FUNCTION_BLOCK RunLifterCelluar EXTENDS RunUnitGeneric
VAR_INPUT
END_VAR
VAR_OUTPUT
END_VAR
VAR	
	//actuator
	//axis
	Axis : POINTER TO RunAxis;
	//cylinder
	Cylinder : POINTER TO RunCylinder;
	
	//lifter
	ptCommandLifterHit : POINTER TO ParameterSet; // raise to hit
	ptCommandLifterRelease : POINTER TO ParameterSet; //release
	ptCommandLifterWorking : POINTER TO ParameterSet; //lift carrier to working position
	//sensor
	ptObstacleSensorStatus : POINTER TO BOOL; //fibers
	ptReachSensorStatus : POINTER TO BOOL; //approximities
	//slot status
	ptPreivousSlotValid : POINTER TO BOOL;
	
END_VAR


CASE State OF
	0:
	//if execute flag on
	bSerialTransition := Axis^.ExecuteParameter(ptBlock:=ptCommandLifterHit);
	1:
	//once reach sensor detected , n
	bSerialTransition := ptReachSensorStatus^;
	2:
	//hold
	bSerialTransition := Cylinder^.Execute(eCylinderCommands.COMMAND_B);
	3:
	//to working position
	bSerialTransition := Axis^.ExecuteParameter(ptCommandLifterWorking);
	4:
	//if release flag on
	bSerialTransition := Axis^.ExecuteParameter(ptCommandLifterHit);
	5:
	//release holder
	bSerialTransition := Cylinder^.Execute(eCylinderCommands.COMMAND_A);
	6:
	IF Axis^.ExecuteParameter(ptCommandLifterRelease) THEN
		NextState := 0;
	END_IF
END_CASE

METHOD CheckReach : BOOL
VAR_INPUT
END_VAR
VAR_OUTPUT
	//neither Done nor Error : Transition
	Done:BOOL;	//successfully
END_VAR
//TODO , slot valid and reach sensor status or not slot valid
Done := ptReachSensorStatus^;
END_METHOD

METHOD FB_init : BOOL
VAR_INPUT
	bInitRetains : BOOL; // if TRUE, the retain variables are initialized (warm start / cold start)
	bInCopyCode : BOOL;  // if TRUE, the instance afterwards gets moved into the copy code (online change)
END_VAR
//initializing , link related commandblock/sensor/cylinder
END_METHOD

METHOD Initialize : BOOL
VAR_INPUT
END_VAR

CASE State OF
	0:
	bSerialTransition:=Cylinder^.Execute(eCylinderCommands.COMMAND_A);
	1:
	IF Axis^.ExecuteParameter(ptCommandLifterRelease) THEN
		NextState := 16#FF;	
	END_IF
END_CASE

Initialize := SUPER^.Initialize(); //call base method
END_METHOD

METHOD RaiseStopper : BOOL
VAR_INPUT
END_VAR
VAR_OUTPUT
	//neither Done nor Error : Transition
	Done:BOOL;	//successfully
END_VAR
VAR
END_VAR
//condition to execute :
//previous slot is valid and
//execute and
//obstacle not existed

//plus my slot is empty
Axis^.ExecuteCommandBlock(
ptBlock:= ptCommandLifterHit, 
execute:= TRUE,//ptPreivousSlotValid^ AND NOT ptObstacleSensorStatus^, 
bufferIndex:=1,
done=> );	

//Done:
//no need to raise
//or need to raise and successfully done	
//Done :=  (ptPreivousSlotValid^ AND ptAxis^.ExecuteCommandBlock.done) OR (NOT ptPreivousSlotValid^);
Done :=done;
END_METHOD

METHOD ReleaseStopper : BOOL
VAR_INPUT
END_VAR
VAR_OUTPUT
	Done:BOOL;	//successfully
END_VAR
Axis^.ExecuteCommandBlock(
ptBlock:= ptCommandLifterRelease, 
execute:= TRUE,//ptPreivousSlotValid^ AND NOT ptObstacleSensorStatus^, 
bufferIndex:=1,
done=> Done);
END_METHOD

END_FUNCTION_BLOCK

(* stored: Version 1.1.0.1, ProductVersion 3.1.4022.10
   POU RunLifterCelluar: Id {8e8fc5f3-47f1-4079-a3ab-596940aadfbf}, SpecialFunc None
   Method CheckReach: Id {67fa871c-5756-49a6-b887-c646b2442d16}
   Method FB_init: Id {a4e43bb3-b045-4468-b1e1-3d38f2c0d86a}
   Method Initialize: Id {21db5a00-f7a1-4530-94de-d799f1b897b9}
   Method RaiseStopper: Id {54b07d97-f47e-4127-8e83-df24e9bcff85}
   Method ReleaseStopper: Id {ed98965b-88bf-4ac2-b044-882d7fe9f646} *)
